TYPE ST_XBox_Controller_Status :
STRUCT
	// Controller's ID
	iControllerNumber  	: INT;
	// Controller is connected to the PC
	bConnected  		: BOOL;
	// Controller is disconnected from the PC
	bDisconnected  		: BOOL;
END_STRUCT
END_TYPE

(* stored: Version 1.1.0.1, ProductVersion 3.1.4024.11
   DUT ST_XBox_Controller_Status: Id {5eb34fdf-0322-4433-adde-2c61be935e0b} *)
